# EPICS substitutions: testApp/Db/userHost.substitutions
# Example substitutions file

file "db/dbExample1.db" {
    { user = "piHost" }
}

file db/dbExample2.db {
    pattern { user, no, scan }
        { "piHost", 1, "1 second" }
        { "piHost", 2, "2 second" }
        { "piHost", 3, "5 second" }
}
